// TIA Portal V15.1 export
// export: Created 2026-01-15T16:29:41.6630389Z, ExportSetting WithDefaults, WithReadOnly, DisplayName Totally Integrated Automation Portal, DisplayVersion V15.1 Update 8, DisplayName TIA Portal Openness, DisplayVersion V15.1 Update 8, DisplayName STEP 7 Professional, DisplayVersion V15.1 Update 8, DisplayName WinCC Advanced, DisplayVersion V15.1 Update 8
FUNCTION_BLOCK "3.RUN_MODE"   // FB3, LAD
{ S7_Optimized_Access := 'TRUE' }
VERSION : 0.1
// stored: AutoNumber false, CodeModifiedDate 2025-08-27T17:11:43.2955348Z, CompileDate 2026-01-15T16:25:55.5692242Z, CreationDate 2026-01-15T16:22:49.8270549Z, DownloadWithoutReinit false, HandleErrorsWithinBlock false, InterfaceModifiedDate 2023-07-24T14:42:19.3789304Z, IsConsistent true, IsIECCheckEnabled false, IsKnowHowProtected false, IsRetainMemResEnabled false, IsWriteProtected false, LibraryConformanceStatus The object is library-conformant., MemoryReserve 100, ModifiedDate 2025-08-27T17:11:43.2955348Z, ParameterModified 2023-07-24T14:41:56.9787559Z, PLCSimAdvancedSupport false, SetENOAutomatically False, StructureModified 2023-07-24T14:42:19.3789304Z, UDAEnableTagReadback false
   VAR_INPUT
      NN_RUN : Bool;
      NN_STOP : Bool;
      SW_SIM : Bool;
      SW_MAN : Bool;
      SW_AUT : Bool;
   END_VAR
   VAR_OUTPUT
      RUN : Bool;
      SIM : Bool;
      MAN : Bool;
      AUT : Bool;
   END_VAR
   VAR
      TEMP1 : Bool;
      TEMP2 : Bool;
   END_VAR
BEGIN

REGION Network 1
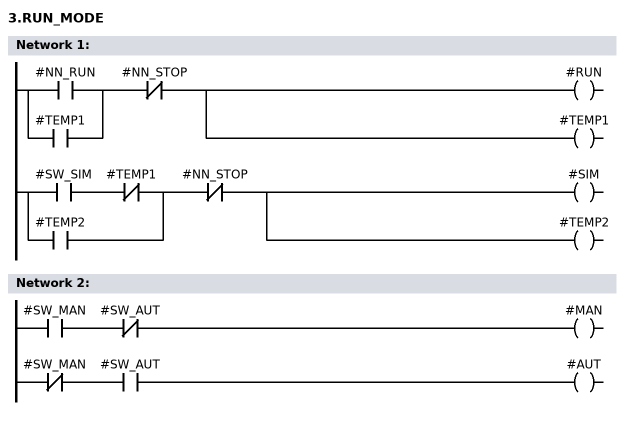
   RUNG wire#powerrail
      Contact( #NN_RUN )
      wire#w1
      I_Contact( #NN_STOP )
      wire#w2
      Coil( #RUN )
   END_RUNG
   RUNG wire#powerrail
      Contact( #TEMP1 )
   END_RUNG wire#w1
   RUNG wire#w2
      Coil( #TEMP1 )
   END_RUNG
   RUNG wire#powerrail
      Contact( #SW_SIM )
      I_Contact( #TEMP1 )
      wire#w3
      I_Contact( #NN_STOP )
      wire#w4
      Coil( #SIM )
   END_RUNG
   RUNG wire#powerrail
      Contact( #TEMP2 )
   END_RUNG wire#w3
   RUNG wire#w4
      Coil( #TEMP2 )
   END_RUNG
   // the same network as SCL:
   #RUN := (#NN_RUN OR #TEMP1) AND NOT #NN_STOP;
   #TEMP1 := #RUN;
   #SIM := ((#SW_SIM AND NOT #TEMP1) OR #TEMP2) AND NOT #NN_STOP;
   #TEMP2 := #SIM;
END_REGION

REGION Network 2
   RUNG wire#powerrail
      Contact( #SW_MAN )
      I_Contact( #SW_AUT )
      Coil( #MAN )
   END_RUNG
   RUNG wire#powerrail
      I_Contact( #SW_MAN )
      Contact( #SW_AUT )
      Coil( #AUT )
   END_RUNG
   // the same network as SCL:
   #MAN := #SW_MAN AND NOT #SW_AUT;
   #AUT := NOT #SW_MAN AND #SW_AUT;
END_REGION
END_FUNCTION_BLOCK
